// TwinCAT 3 PLC project Testprojekt
// ProgramVersion: 3.1.4026.1+5afe9138fb3b9c21507bc48985af5a0bc4d3d11a
// libraries:
//   Tc2_Standard, * (Beckhoff Automation GmbH)
//   Tc2_System, * (Beckhoff Automation GmbH)
// project tree:
//   / PlcTask.TcTTO
//   POUs/ MAIN.TcPOU

CONFIGURATION Testprojekt
    RESOURCE PLC ON TwinCAT3
        TASK PlcTask(INTERVAL := T#10ms, PRIORITY := 20);
        PROGRAM MAIN WITH PlcTask : MAIN;
    END_RESOURCE
END_CONFIGURATION

// ---- POUs/MAIN.TcPOU
PROGRAM MAIN
VAR
	Ialive : Int;
END_VAR

Ialive := Ialive + 1;

END_PROGRAM
